{attribute 'qualified_only'}
VAR_GLOBAL
	
	bRunningLight : BOOL;
	rCylinderVel : REAL;
	rCylinderPos : REAL;
	


	
END_VAR

(* stored: Version 1.1.0.1, ProductVersion 3.1.4024.10
   GVL output: Id {fc17bddc-aa60-41d3-a681-bfb85a0ae552} *)
